TYPE ST_INPUTS_Strainer:
STRUCT
	
	Mode:     	E_DeviceMode;
	Command:     E_DeviceState;

END_STRUCT
END_TYPE

(* stored: Version 1.1.0.1, ProductVersion 3.1.4024.12
   DUT ST_INPUTS_Strainer: Id {25a66251-a79a-43da-be33-4b7e8d1799ab} *)
